PROGRAM MAIN
VAR
	aEvents : ARRAY[1..100] OF ST_Event;
	sTempString : STRING(255);
END_VAR

sTempString := aEvents[33].sEventText;

END_PROGRAM

(* stored: Version 1.1.0.1, ProductVersion 3.1.4024.11
   POU MAIN: Id {46b87271-a47f-40d1-9e75-510d5206adec}, SpecialFunc None *)
